FUNCTION "FC_RouteFSM" : Void
{ S7_Optimized_Access := 'TRUE' }
VERSION : 4.6
// ==============================================================================
// FC_RouteFSM - Керування маршрутом (Mailbox Pattern v4.0)
// ==============================================================================
// Версія: 4.6.0
// Дата: 2026-05-15
// ==============================================================================
// ЗМІНИ v4.6.0:
//   [FEAT] Реалізовано "Різкий останов" (Fast Stop) при аварії механізму.
//   [FEAT] Додана детальна перевірка GrainType для ям та силосів.
//   [FIX] Виключено перевірку типу для конкретних силосів (1,2,19,25,26,27).
//   [FEAT] Додано очікування цільової позиції для засувок (Gate2P) та клапанів (Valve3P).
//   [FEAT] Додано очікування цільової позиції для засувок (Gate2P) та клапанів (Valve3P) при пуску та зупинці.
//   [FIX] Виправлено назву константи TYPE_RECEIVING_PIT.
//
// ЗМІНИ v4.0.0:
//   [FIX] RUNNING/STOPPING: затримка (StartDelayMs/StopDelayMs) тепер відбувається
//         ПЕРЕД видачею команди, а не ПІСЛЯ досягнення цільового стану.
//         БУЛО: CMD_START → wait target → IF delay > 0 → pause → advance
//         СТАЛО: IF delay > 0 → pause first → CMD_START → wait target → advance
//         stepPauseTck = 0 означає "новий крок, затримка ще не почалась".
//   [FEAT] Додано підтримку TYPE_FAN та TYPE_FEEDER в CASE для читання затримок.
//   [FIX] Видалено використання RS_TimeoutMs (якого більше немає в UDT_RouteStep).
//         Тепер використовуються індивідуальні затримки з механізмів.
//
// ЗМІНИ v3.9.2:
//   [FIX] STOPPING: advance-блок переписано з явним флагом doAdvance (VAR_TEMP).
//         БУЛО: окремий "NOT stepPause AND stopped" блок — умова могла бути TRUE
//               в циклах де pause ще не виставлена.
//         СТАЛО: doAdvance := TRUE ТІЛЬКИ у двох явних випадках:
//               - Phase A: механізм зупинився AND RS_TimeoutMs = 0
//               - Phase B: таймер спрацював (timeElapsed = TRUE)
//         Симетрично з RUNNING (де advance теж всередині Phase B IF timeElapsed).
//
// ЗМІНИ v3.9.1:
//   [FIX] TIA Portal SCL не дозволяє виклик функції з VAR_OUTPUT в IF-виразі.
//         FC_TimeElapsedMs (має VAR_OUTPUT ElapsedMs, NowTck) → результат
//         тепер зберігається у VAR_TEMP timeElapsed : BOOL перед IF.
//         Додано VAR_TEMP секцію.
//
// ЗМІНИ v3.9.0:
//   [FEAT-3] RUNNING: пауза між кроками через RS_TimeoutMs (аналогічно STOPPING).
//            Фаза A: видати команду → чекаємо цільового стану (RUNNING або IDLE).
//            Фаза B (stepPause=TRUE): чекаємо RS_TimeoutMs мс, потім advance.
//            RS_TimeoutMs = 0 → Фаза B відсутня (поведінка як раніше).
//            Перейменовано: stopPause→stepPause, stopPauseTck→stepPauseTck.
//
// ЗМІНИ v3.8.0:
//   [FEAT-2] STOPPING: пауза між кроками через RS_TimeoutMs.
//            Фаза A: CMD_STOP кожен цикл → чекаємо зупинки механізму.
//            Фаза B (stepPause=TRUE): чекаємо RS_TimeoutMs мс після зупинки.
//            RS_TimeoutMs = 0 → Фаза B відсутня (поведінка як у v3.7).
//            Нові поля UDT_RouteFsm: stepPause : BOOL, stepPauseTck : DINT.
//
// ЗМІНИ v3.7.0:
//   [FEAT-1] STOPPING: послідовна зупинка у зворотньому порядку.
//            БУЛО: CMD_STOP до всіх механізмів одночасно (FOR по всіх кроках),
//                  потім очікування allStopped.
//            СТАЛО: зупинка крок-за-кроком від stepCnt до 1 (1-based).
//                   Кожен цикл — CMD_STOP до поточного кроку (RF_ActiveStep).
//                   Коли поточний зупинився → RF_ActiveStep-- → наступний крок.
//                   Коли крок 1 зупинився → CMD_RELEASE_OWNER для всіх → ABORTED.
//            RF_ActiveStep ініціалізується = stepCnt при вході з RUNNING (1-based).
//
// ЗМІНИ v3.6.2:
//   [FIX-12] VALIDATING: додано перевірку сумісності RS_Action + RS_Wait.
//            RS_ACT_STOP + RS_WAIT_RUNNING → ROUTE_REJ_BY_CONTRACT.
//            До виправлення: ця комбінація проходила валідацію, але у RUNNING
//            механізм після CMD_STOP ніколи не досягав STS_RUNNING →
//            крок зависав нескінченно (до зовнішнього fault або SafetyStop).
//
// ЗМІНИ v3.6.1:
//   [FIX-10] Ранній скан anyFault/anyLocal + GlobalSafetyStop блок:
//            додано IF slot > MECHS_COUNT THEN CONTINUE перед Mechs[slot].
//            До виправлення: у першому циклі нової команди з невалідним RS_Slot
//            обидва цикли зверталися до Mechs[invalid] до того, як VALIDATING
//            встигав відхилити крок → потенційний OOB і зупинка CPU (OB121).
//
// ЗМІНИ v3.6.0:
//   [FIX-8] Виправлено хибний коментар у STOPPING → CMD_RELEASE_OWNER.
//           БУЛО:   "STS_DISABLED → OwnerCur вже NONE → ARB_OWNER_BUSY"
//           ФАКТ:   OwnerCur залишається OWNER_ROUTE після переходу у STS_DISABLED
//                   (механізм не скидає OwnerCur самостійно).
//                   CMD_RELEASE_OWNER → ARB_WRONG_STATUS (DISABLED ≠ IDLE/FAULT).
//                   dummyOk → ABORTED → retry кожен цикл → Enable_OK відновлено
//                   → STS_IDLE → ARB_OK → звільнено ✓   (FIX-5 зберігає StepCount).
//
//   [FIX-9] Видалено недосяжний код у VALIDATING (перевірка startEdge).
//           startEdge завжди FALSE у циклі VALIDATING:
//             Цикл N (IDLE):       lastCmd=RT_CMD_NONE → startEdge=TRUE → lastCmd:=RT_CMD_START
//             Цикл N+1 (VALID.):   lastCmd=RT_CMD_START, Cmd=RT_CMD_START → startEdge=FALSE
//           Supervisor блокує новий START поки isActive → RouteExecutor не змінюється.
//           Константа ROUTE_REJ_DUPLICATE_START більше не використовується.
//
// ЗМІНИ v3.5.0:
//   [FIX-7] ABORTED/REJECTED: startEdge → прямий перехід у VALIDATING.
//
//           ПРОБЛЕМА: маршрут у ABORTED, SCADA надсилає RT_CMD_START.
//           Цикл N:   Supervisor копіює START → RouteExecutor (processedRouteId захищає).
//                     FSM ABORTED: RC_Cmd ≠ RT_CMD_NONE → лишається ABORTED.
//           Цикл N+1: Cleanup бачить ABORTED + allReleased → RC_Cmd=RT_CMD_NONE, StepCount=0.
//                     FSM ABORTED: RT_CMD_NONE → IDLE.
//           Цикл N+2: FSM IDLE: RC_Cmd=RT_CMD_NONE → startEdge=FALSE → нічого.
//           START мовчки загублено.
//
//           РІШЕННЯ: у ABORTED/REJECTED перевіряємо startEdge першим.
//           Якщо startEdge → VALIDATING (скидаємо ResultCode/ActiveStep/StepSts).
//           Цикл N+1: стан вже VALIDATING → Cleanup не чіпає → кроки збережені ✓
//           Механізми ще OWNER_ROUTE (ABORTED-retry) → VALIDATING відкидає REJ_BY_OWNER
//           (коректна поведінка; оператор бачить REJECTED, а не мовчазний IDLE).
//
// ЗМІНИ v3.4.0:
//   - VALIDATING: додано перевірку RS_Slot > MECHS_COUNT → ROUTE_REJ_BY_CONTRACT.
//   - Захист від виходу за межі масиву Mechs[] при невалідному слоті від SCADA.
//   - Перевірка стоїть першою у циклі — до будь-якого звернення до Mechs[slot].
//   - Всі наступні стани (STARTING/RUNNING/STOPPING) отримують гарантовано валідний слот.
//
// ==============================================================================
// ЗМІНИ v3.0.0:
//   - FC_ArbiterMech: повертає USINT (RejectCode) замість BOOL
//   - CMD_NONE заборонено → CMD_SET_OWNER_SCADA / CMD_RELEASE_OWNER
//   - lockOkOne, cmdOk, dummyOk: BOOL → USINT у UDT_RouteFsm
//
// ЗМІНИ v3.1.0:
//   - ABORTED: retry CMD_RELEASE_OWNER кожен цикл поки OwnerCur = OWNER_ROUTE
//   - Вирішує застряглий ownership після GlobalSafetyStop
//
// ЗМІНИ v3.2.0:
//   - STOPPING: виправлено allStopped — рахує STS_FAULT/DISABLED/LOCAL як зупинені
//   - БУЛО:   Status <> STS_IDLE → не зупинений
//   - СТАЛО:  Status IN {STARTING, RUNNING, STOPPING} → не зупинений
//
// ЗМІНИ v3.3.0:
//   - GlobalSafetyStop: ДОДАНО CMD_STOP перед CMD_RELEASE_OWNER
//   - БУЛО: тільки CMD_RELEASE_OWNER (best effort) → мотор міг крутитись ~2 сек
//   - СТАЛО: спочатку CMD_STOP (наказ зупинитись), потім CMD_RELEASE_OWNER
//   - Тепер механізм отримує команду зупинки негайно і йде STS_STOPPING→STS_IDLE
//     замість чекати SpeedLost timeout → STS_FAULT
//   - CMD_RELEASE_OWNER після CMD_STOP все одно може повернути ARB_WRONG_STATUS
//     (механізм ще RUNNING/STOPPING), retry відбувається у ABORTED як раніше
//
// ГАРАНТІЇ ЗУПИНКИ:
//   Нормальний STOP_OP:
//     STOPPING: CMD_STOP кожен цикл → STS_STOPPING→STS_IDLE →
//     allStopped → CMD_RELEASE_OWNER (ARB_OK) → ABORTED ✓
//
//   Аварія під час зупинки (STOPPING):
//     STS_FAULT → allStopped (FAULT рахується) →
//     CMD_RELEASE_OWNER (ARB_OK, FAULT дозволено) → ABORTED ✓
//
//   Enable_OK знімається під час зупинки (STOPPING):
//     STS_DISABLED + OwnerCur=NONE (механізм сам скинув) → allStopped →
//     CMD_RELEASE_OWNER → ARB_OWNER_BUSY (dummyOk) → ABORTED ✓
//
//   GlobalSafetyStop (механізм у STS_RUNNING):
//     CMD_STOP → Mechs[slot].Cmd=CMD_STOP → механізм → STS_STOPPING
//     CMD_RELEASE_OWNER → ARB_WRONG_STATUS (ще не IDLE) → ABORTED
//     Retry у ABORTED: STS_STOPPING→STS_IDLE → ARB_OK → OwnerCur=NONE ✓
//     (якщо апаратна безпека вбила живлення → STS_FAULT → ARB_OK ✓)
//
// АРХІТЕКТУРА:
//   FC_RouteFSM    — логіка переходів, послідовність кроків
//   FC_ArbiterMech — захоплення ownership, запис команди
//   FC_Noria/...   — виконання команди, зміна Status, аварії
//   FC_Route_Supervisor — Mailbox→RouteExecutor, виклик FSM, cleanup
// ==============================================================================
   VAR_INPUT
      RouteIdx : USInt;   // ID маршруту (1..12)
      Cmd : "UDT_RouteCmd";   // Команда та кроки маршруту
   END_VAR

   VAR_OUTPUT
      Sts : "UDT_RouteStatus";
   END_VAR

   VAR_IN_OUT
      Mechs : Array[0.."MECHS_COUNT"] of "UDT_BaseMechanism";
      Fsm : "UDT_RouteFsm";
   END_VAR

   VAR_TEMP
      timeElapsed : Bool;   // проміжний результат FC_TimeElapsedMs
      elapsedMs : DInt;   // допоміжний вихід FC_TimeElapsedMs (ігнорується)
      nowTck : DInt;   // допоміжний вихід FC_TimeElapsedMs (ігнорується)
      doAdvance : Bool;   // TRUE = виконати advance у STOPPING (після Phase A або Phase B)
      stepDelayMs : DInt;   // індивідуальна затримка з механізму (StartDelayMs/StopDelayMs)
      grainTypePit : Int;   // тип зерна ями (для перевірки сумісності)
      grainTypeSilo : Int;   // тип зерна силосу (для перевірки сумісності)
      firstSiloGrainType : Int;   // тип першого силосу в маршруті
      siloCnt : Int;   // кількість силосів у маршрутi
      siloMissingType : Bool;   // TRUE = один із силосів має незаданий тип
      siloGrainMismatch : Bool;   // TRUE = в маршруті два силоси з різними типами зерна
      isSiloExcluded : Bool;   // TRUE = силос виключений з перевірки GrainType
      forceGrainType : Bool;   // TRUE = силос має Force_Code BIT10 — ігнорувати перевірку GrainType
      hasPit : Bool;   // TRUE = у маршруті є яма
      hasSilo : Bool;   // TRUE = у маршруті є силос
   END_VAR


BEGIN

	// =========================================================
	// Edge detection команд маршруту
	// =========================================================
	#Fsm.startEdge := (#Cmd.RC_Cmd = "RT_CMD_START") AND (#Fsm.lastCmd <> "RT_CMD_START");
	#Fsm.stopOpEdge := (#Cmd.RC_Cmd = "RT_CMD_STOP_OP") AND (#Fsm.lastCmd <> "RT_CMD_STOP_OP");
	#Fsm.lastCmd := #Cmd.RC_Cmd;

	// =========================================================
	// Кількість кроків (з обмеженням)
	// =========================================================
	#Fsm.stepCnt := USINT_TO_INT(#Cmd.RC_StepCount);
	IF #Fsm.stepCnt < 1 THEN
	    #Fsm.stepCnt := 1;
	END_IF;
	IF #Fsm.stepCnt > "ROUTE_MAX_STEPS" THEN
	    #Fsm.stepCnt := "ROUTE_MAX_STEPS";
	END_IF;

	// Захист від неініціалізованого стану
	IF #Fsm.RF_State = 0 THEN
	    #Fsm.RF_State := "ROUTE_STS_IDLE";
	END_IF;

	// =========================================================
	// Сканування механізмів: аварії та LocalManual
	// =========================================================
	#Fsm.anyFault := FALSE;
	#Fsm.anyLocal := FALSE;
	#Fsm.safetyHit := FALSE;

	IF #Fsm.stepCnt > 0 THEN
	    FOR #Fsm.i := 1 TO #Fsm.stepCnt DO
	        #Fsm.slot := #Cmd.RC_Steps[#Fsm.i].RS_Slot;
	        IF #Fsm.slot > "MECHS_COUNT" THEN
	            CONTINUE;
	        END_IF;

	        IF #Mechs[#Fsm.slot].FLTCode <> 0 THEN
	            #Fsm.anyFault := TRUE;
	        END_IF;

	        IF "GlobalLocalManual" OR #Mechs[#Fsm.slot].LocalManual THEN
	            #Fsm.anyLocal := TRUE;
	        END_IF;

	        IF #Fsm.anyFault AND #Fsm.anyLocal THEN
	            EXIT;
	        END_IF;
	    END_FOR;
	END_IF;

	// =========================================================
	// АВАРІЙНА ЗУПИНКА (GlobalSafetyStop) — найвищий пріоритет
	// =========================================================
	// Послідовність для кожного механізму:
	//   1. CMD_STOP       — наказ зупинитись негайно (незалежно від послідовності)
	//                       ARB_OK → Mechs[slot].Cmd = CMD_STOP ✓
	//                       ARB_OWNER_BUSY → не наш механізм, не критично
	//                       ARB_LOCAL_MANUAL → оператор сам відповідає
	//   2. CMD_RELEASE_OWNER — спроба звільнити власника (best effort)
	//                       ARB_WRONG_STATUS якщо ще RUNNING/STOPPING → retry у ABORTED
	//
	// Чому не чекаємо STS_IDLE перед CMD_RELEASE_OWNER:
	//   Safety stop = негайно, без очікування. Механізм зупиниться сам
	//   (STS_STOPPING→STS_IDLE або апаратна безпека→STS_FAULT).
	//   Retry у ABORTED звільнить ownership коли механізм зупиниться.
	// =========================================================
	IF "GlobalSafetyStop" THEN
	    #Fsm.safetyHit := TRUE;

	    IF #Fsm.stepCnt > 0 THEN
	        FOR #Fsm.i := 1 TO #Fsm.stepCnt DO
	            #Fsm.slot := #Cmd.RC_Steps[#Fsm.i].RS_Slot;
	            IF #Fsm.slot > "MECHS_COUNT" THEN
	                CONTINUE;
	            END_IF;

	            // КРОК 1: Зупинити механізм
	            #Fsm.dummyOk := "FC_ArbiterMech"(
	                                             OwnerReq := "OWNER_ROUTE",
	                                             OwnerReqId := USINT_TO_UINT(#RouteIdx),
	                                             ReqCmd := "CMD_STOP",
	                                             ReqParam1 := 0,
	                                             M := #Mechs[#Fsm.slot]
	            );

	            // КРОК 2: Звільнити власника (best effort)
	            // Якщо STS_RUNNING/STOPPING → ARB_WRONG_STATUS → retry у ABORTED
	            #Fsm.dummyOk := "FC_ArbiterMech"(
	                                             OwnerReq := "OWNER_ROUTE",
	                                             OwnerReqId := USINT_TO_UINT(#RouteIdx),
	                                             ReqCmd := "CMD_RELEASE_OWNER",
	                                             ReqParam1 := 0,
	                                             M := #Mechs[#Fsm.slot]
	            );

	        END_FOR;
	    END_IF;

	    #Fsm.RF_State := "ROUTE_STS_ABORTED";
	    #Fsm.RF_ResultCode := "ROUTE_ABRT_BY_SAFETY";
	END_IF;

	// =========================================================
	// FSM маршруту
	// =========================================================
	IF NOT #Fsm.safetyHit THEN

	    // --------------------------------------------------------
	    // IDLE
	    // --------------------------------------------------------
	    IF #Fsm.RF_State = "ROUTE_STS_IDLE" THEN

	        IF #Fsm.startEdge THEN
	            #Fsm.RF_ResultCode := 0;
	            #Fsm.RF_AbortLatched := 0;
	            #Fsm.RF_ActiveStep := 1;  // 1-based: перший крок [1]
	            #Fsm.RF_StepSts := "STEP_STS_IDLE";
	            #Fsm.RF_State := "ROUTE_STS_VALIDATING";
	        END_IF;

	        // --------------------------------------------------------
	        // VALIDATING
	        // --------------------------------------------------------
	    ELSIF #Fsm.RF_State = "ROUTE_STS_VALIDATING" THEN

	        IF #Fsm.stepCnt <= 0 THEN
	            #Fsm.RF_State := "ROUTE_STS_REJECTED";
	            #Fsm.RF_ResultCode := "ROUTE_REJ_BY_CONTRACT";

	        ELSE
	            FOR #Fsm.i := 1 TO #Fsm.stepCnt DO
	                #Fsm.slot := #Cmd.RC_Steps[#Fsm.i].RS_Slot;
	                #Fsm.stepOk := TRUE;

	                // Сушилка не керується маршрутом — скіп
	                IF #Fsm.slot <= "MECHS_COUNT" THEN
	                    IF #Mechs[#Fsm.slot].DeviceType = "TYPE_SUSHKA" THEN
	                        CONTINUE;
	                    END_IF;
	                END_IF;

	                // Контракт: RS_Slot (перша перевірка — до будь-якого Mechs[slot])
	                IF #Fsm.slot > "MECHS_COUNT" THEN
	                    #Fsm.stepOk := FALSE;
	                END_IF;

	                // Контракт: RS_Action
	                IF (#Cmd.RC_Steps[#Fsm.i].RS_Action <> "RS_ACT_START")
	                    AND (#Cmd.RC_Steps[#Fsm.i].RS_Action <> "RS_ACT_STOP") THEN
	                    #Fsm.stepOk := FALSE;
	                END_IF;

	                // Контракт: RS_Wait
	                IF (#Cmd.RC_Steps[#Fsm.i].RS_Wait <> "RS_WAIT_RUNNING")
	                    AND (#Cmd.RC_Steps[#Fsm.i].RS_Wait <> "RS_WAIT_STOPPED") THEN
	                    #Fsm.stepOk := FALSE;
	                END_IF;

	                // Контракт: RS_Action + RS_Wait сумісність
	                // RS_ACT_STOP + RS_WAIT_RUNNING: після CMD_STOP механізм іде
	                // STOPPING→IDLE і ніколи не повернеться у STS_RUNNING →
	                // крок ніколи не завершиться → маршрут зависає в RUNNING.
	                IF (#Cmd.RC_Steps[#Fsm.i].RS_Action = "RS_ACT_STOP")
	                    AND (#Cmd.RC_Steps[#Fsm.i].RS_Wait = "RS_WAIT_RUNNING") THEN
	                    #Fsm.stepOk := FALSE;
	                END_IF;

	                IF NOT #Fsm.stepOk THEN
	                    #Fsm.RF_State := "ROUTE_STS_REJECTED";
	                    #Fsm.RF_ResultCode := "ROUTE_REJ_BY_CONTRACT";
	                    EXIT;

	                ELSIF #Mechs[#Fsm.slot].OwnerCur <> "OWNER_NONE" THEN
	                    #Fsm.RF_State := "ROUTE_STS_REJECTED";
	                    #Fsm.RF_ResultCode := "ROUTE_REJ_BY_OWNER";
	                    EXIT;

	                ELSIF (NOT #Mechs[#Fsm.slot].Enable_OK)
	                    OR "GlobalLocalManual"
	                    OR #Mechs[#Fsm.slot].LocalManual
	                    OR (#Mechs[#Fsm.slot].FLTCode <> 0) THEN
	                    #Fsm.RF_State := "ROUTE_STS_REJECTED";
	                    #Fsm.RF_ResultCode := "ROUTE_REJ_NOT_READY";
	                    EXIT;
	                END_IF;

	            END_FOR;

	            IF #Fsm.RF_State = "ROUTE_STS_VALIDATING" THEN
	                // Перевірка GrainType: яма і силос повинні мати однаковий ненульовий тип,
	                // а якщо в маршруті два силоси — їхні типи також повинні співпадати.
	                #grainTypePit := 0;
	                #grainTypeSilo := 0;
	                #firstSiloGrainType := 0;
	                #siloCnt := 0;
	                #siloMissingType := FALSE;
	                #siloGrainMismatch := FALSE;
	                #isSiloExcluded := FALSE;
	                #forceGrainType := FALSE;
	                #hasPit := FALSE;
	                #hasSilo := FALSE;

	                FOR #Fsm.i := 1 TO #Fsm.stepCnt DO
	                    #Fsm.slot := #Cmd.RC_Steps[#Fsm.i].RS_Slot;
	                    IF #Fsm.slot <= "MECHS_COUNT" THEN
	                        IF #Mechs[#Fsm.slot].DeviceType = "TYPE_RECEIVING_PIT" THEN
	                            #hasPit := TRUE;
	                            #grainTypePit := "DB_Mechs".ReceivingPit[#Mechs[#Fsm.slot].TypedIndex].GrainType;
	                        ELSIF #Mechs[#Fsm.slot].DeviceType = "TYPE_SILOS" THEN
	                            #hasSilo := TRUE;
	                            // Исключения: силосы с TypedIndex 1,2,19,25,26,27 не проверяем GrainType
	                            #isSiloExcluded := (#Mechs[#Fsm.slot].TypedIndex = 1 OR #Mechs[#Fsm.slot].TypedIndex = 2 OR
	                            #Mechs[#Fsm.slot].TypedIndex = 19 OR #Mechs[#Fsm.slot].TypedIndex = 25 OR
	                            #Mechs[#Fsm.slot].TypedIndex = 26 OR #Mechs[#Fsm.slot].TypedIndex = 27);
	                            IF NOT #isSiloExcluded THEN
	                                #siloCnt := #siloCnt + 1;
	                                #grainTypeSilo := "DB_Mechs".Silos[#Mechs[#Fsm.slot].TypedIndex].GrainType;
	                                IF #grainTypeSilo = 0 THEN
	                                    #siloMissingType := TRUE;
	                                END_IF;
	                                IF #siloCnt = 1 THEN
	                                    #firstSiloGrainType := #grainTypeSilo;
	                                ELSIF #firstSiloGrainType <> #grainTypeSilo THEN
	                                    #siloGrainMismatch := TRUE;
	                                END_IF;
	                            END_IF;
	                            IF (#Mechs[#Fsm.slot].Force_Code AND 1024) <> 0 THEN
	                                #forceGrainType := TRUE;
	                            END_IF;
	                        END_IF;
	                    END_IF;
	                END_FOR;

	                IF NOT #forceGrainType THEN
	                    // Силос в маршруті і один із силосів не має заданого типу
	                    IF #hasSilo AND #siloMissingType THEN
	                        #Fsm.RF_State := "ROUTE_STS_REJECTED";
	                        #Fsm.RF_ResultCode := "ROUTE_REJ_GRAIN_NOT_SET";
	                        // Яма в маршруті і її тип = 0
	                    ELSIF #hasPit AND #grainTypePit = 0 THEN
	                        #Fsm.RF_State := "ROUTE_STS_REJECTED";
	                        #Fsm.RF_ResultCode := "ROUTE_REJ_GRAIN_NOT_SET";
	                        // Два силоси в маршруті і їхні типи не співпадають
	                    ELSIF #siloGrainMismatch THEN
	                        #Fsm.RF_State := "ROUTE_STS_REJECTED";
	                        #Fsm.RF_ResultCode := "ROUTE_REJ_SILOS_GRAIN_MISMATCH";
	                        // Обидва (яма + силос) в маршруті і типи не співпадають
	                    ELSIF #hasSilo AND #hasPit AND #firstSiloGrainType <> #grainTypePit THEN
	                        #Fsm.RF_State := "ROUTE_STS_REJECTED";
	                        #Fsm.RF_ResultCode := "ROUTE_REJ_GRAIN_MISMATCH";
	                    END_IF;
	                END_IF;
	            END_IF;

	            IF #Fsm.RF_State = "ROUTE_STS_VALIDATING" THEN
	                #Fsm.RF_State := "ROUTE_STS_STARTING";
	            END_IF;
	        END_IF;

	        // --------------------------------------------------------
	        // STARTING — атомарне захоплення всіх механізмів
	        // --------------------------------------------------------
	    ELSIF #Fsm.RF_State = "ROUTE_STS_STARTING" THEN

	        #Fsm.lockOkAll := TRUE;

	        IF #Fsm.stepCnt > 0 THEN
	            FOR #Fsm.i := 1 TO #Fsm.stepCnt DO
	                #Fsm.slot := #Cmd.RC_Steps[#Fsm.i].RS_Slot;

	                // Сушилка не керується маршрутом — не захоплюємо owner
	                IF #Mechs[#Fsm.slot].DeviceType = "TYPE_SUSHKA" THEN
	                    CONTINUE;
	                END_IF;

	                // CMD_SET_OWNER_SCADA = захопити власника без виконання команди
	                #Fsm.lockOkOne := "FC_ArbiterMech"(
	                                                   OwnerReq := "OWNER_ROUTE",
	                                                   OwnerReqId := USINT_TO_UINT(#RouteIdx),
	                                                   ReqCmd := "CMD_SET_OWNER_SCADA",
	                                                   ReqParam1 := 0,
	                                                   M := #Mechs[#Fsm.slot]
	                );

	                IF #Fsm.lockOkOne <> "ARB_OK" THEN
	                    #Fsm.lockOkAll := FALSE;
	                END_IF;
	            END_FOR;
	        ELSE
	            #Fsm.lockOkAll := FALSE;
	        END_IF;

	        IF NOT #Fsm.lockOkAll THEN
	            // Відкат: звільнити вже захоплені механізми.
	            // Механізми ще у IDLE (не запускались) → CMD_RELEASE_OWNER пройде.
	            // Механізм що не захопився → ARB_OWNER_BUSY → dummyOk.
	            IF #Fsm.stepCnt > 0 THEN
	                FOR #Fsm.i := 1 TO #Fsm.stepCnt DO
	                    #Fsm.slot := #Cmd.RC_Steps[#Fsm.i].RS_Slot;

	                    #Fsm.dummyOk := "FC_ArbiterMech"(
	                                                     OwnerReq := "OWNER_ROUTE",
	                                                     OwnerReqId := USINT_TO_UINT(#RouteIdx),
	                                                     ReqCmd := "CMD_RELEASE_OWNER",
	                                                     ReqParam1 := 0,
	                                                     M := #Mechs[#Fsm.slot]
	                    );
	                END_FOR;
	            END_IF;

	            #Fsm.RF_State := "ROUTE_STS_REJECTED";
	            #Fsm.RF_ResultCode := "ROUTE_REJ_BY_OWNER";

	        ELSE
	            #Fsm.RF_State := "ROUTE_STS_RUNNING";
	        END_IF;

	        // --------------------------------------------------------
	        // RUNNING — виконання кроків по черзі (затримка ПЕРЕД командою)
	        // --------------------------------------------------------
	    ELSIF #Fsm.RF_State = "ROUTE_STS_RUNNING" THEN

	        // --- Умови переривання (перевіряються до виконання кроку) ---
	        IF #Fsm.stopOpEdge THEN
	            #Fsm.RF_AbortLatched := "ROUTE_ABRT_BY_OPERATOR";
	            #Fsm.RF_ActiveStep := INT_TO_USINT(#Fsm.stepCnt);  // 1-based: останній крок [stepCnt]
	            #Fsm.stepPause := FALSE;
	            #Fsm.stepPauseTck := 0;
	            #Fsm.RF_State := "ROUTE_STS_STOPPING";

	        ELSIF #Fsm.anyLocal THEN
	            #Fsm.RF_AbortLatched := "ROUTE_ABRT_BY_LOCAL";
	            #Fsm.RF_ActiveStep := INT_TO_USINT(#Fsm.stepCnt);  // 1-based
	            #Fsm.stepPause := FALSE;
	            #Fsm.stepPauseTck := 0;
	            #Fsm.RF_State := "ROUTE_STS_STOPPING";

	        ELSIF #Fsm.anyFault THEN
	            #Fsm.RF_ResultCode := "ROUTE_ABRT_BY_FAULT";

	            // РЕЗКИЙ ОСТАНОВ: негайно зупинити всі механізми маршруту
	            IF #Fsm.stepCnt > 0 THEN
	                FOR #Fsm.i := 1 TO #Fsm.stepCnt DO
	                    #Fsm.slot := #Cmd.RC_Steps[#Fsm.i].RS_Slot;
	                    IF #Fsm.slot > 0 AND #Fsm.slot <= "MECHS_COUNT" THEN
	                        #Fsm.dummyOk := "FC_ArbiterMech"(
	                            OwnerReq := "OWNER_ROUTE",
	                            OwnerReqId := USINT_TO_UINT(#RouteIdx),
	                            ReqCmd := "CMD_STOP",
	                            ReqParam1 := 0,
	                            M := #Mechs[#Fsm.slot]);
	                    END_IF;
	                END_FOR;
	            END_IF;
	            #Fsm.RF_State := "ROUTE_STS_ABORTED";

	        ELSE
	            // --- Поточний крок ---
	            #Fsm.stepIdx := USINT_TO_INT(#Fsm.RF_ActiveStep);

	            IF #Fsm.stepIdx > #Fsm.stepCnt THEN
	                // Всі кроки виконано — залишаємось у RUNNING.
	                // Механізми залишаються під Owner=ROUTE.
	                // SCADA бачить ResultCode=200 → маршрут активний.
	                #Fsm.RF_ResultCode := "ROUTE_OK_RUNNING";  // BIT15 = 32768

	            ELSE
	                #Fsm.slot := #Cmd.RC_Steps[#Fsm.stepIdx].RS_Slot;

	                // === Читати StartDelayMs з механизма ===
	                CASE #Mechs[#Fsm.slot].DeviceType OF
	                    "TYPE_REDLER":
	                        #stepDelayMs := "DB_Mechs".Redler[#Mechs[#Fsm.slot].TypedIndex].StartDelayMs;
	                    "TYPE_NORIA":
	                        #stepDelayMs := "DB_Mechs".Noria[#Mechs[#Fsm.slot].TypedIndex].StartDelayMs;
	                    "TYPE_SEPARATOR":
	                        #stepDelayMs := "DB_Mechs".Separator[#Mechs[#Fsm.slot].TypedIndex].StartDelayMs;
	                    "TYPE_FAN":
	                        #stepDelayMs := "DB_Mechs".Fan[#Mechs[#Fsm.slot].TypedIndex].StartDelayMs;
	                    "TYPE_FEEDER":
	                        #stepDelayMs := "DB_Mechs".Feeder[#Mechs[#Fsm.slot].TypedIndex].StartDelayMs;
	                    ELSE
	                        #stepDelayMs := 0;
	                END_CASE;

	                // === Фаза: Затримка ПЕРЕД командою ===
	                IF #stepDelayMs > 0 AND #Fsm.stepPauseTck = 0 AND NOT #Fsm.stepPause THEN
	                    #timeElapsed := "FC_TimeElapsedMs"(
	                                                       StartTck := 0,
	                                                       TimeoutMs := 0,
	                                                       ElapsedMs => #elapsedMs,
	                                                       NowTck => #Fsm.stepPauseTck);
	                    #Fsm.stepPause := TRUE;
	                END_IF;

	                IF #Fsm.stepPause THEN
	                    // Чекаємо завершення затримки ПЕРЕД командою
	                    #timeElapsed := "FC_TimeElapsedMs"(
	                                                       StartTck := #Fsm.stepPauseTck,
	                                                       TimeoutMs := #stepDelayMs,
	                                                       ElapsedMs => #elapsedMs,
	                                                       NowTck => #nowTck);
	                    IF #timeElapsed THEN
	                        #Fsm.stepPause := FALSE;
	                    END_IF;
	                END_IF;

	                // === Сушилка: скіп кроку ===
	                IF #Mechs[#Fsm.slot].DeviceType = "TYPE_SUSHKA" THEN
	                    #Fsm.stepPauseTck := 0;
	                    #Fsm.RF_ActiveStep := #Fsm.RF_ActiveStep + 1;
	                    #Fsm.RF_StepSts := "STEP_STS_DONE";
	                ELSE
	                // === Фаза: Видача команди + очікування цілі ===
	                IF NOT #Fsm.stepPause THEN
	                    // Видати команду поточного кроку через арбітр (кожен цикл)
	                    IF #Cmd.RC_Steps[#Fsm.stepIdx].RS_Action = "RS_ACT_START" THEN
	                        #Fsm.cmdOk := "FC_ArbiterMech"(
	                                                       OwnerReq := "OWNER_ROUTE",
	                                                       OwnerReqId := USINT_TO_UINT(#RouteIdx),
	                                                       ReqCmd := "CMD_START",
	                                                       ReqParam1 := #Cmd.RC_Steps[#Fsm.stepIdx].RS_StartParam,
	                                                       M := #Mechs[#Fsm.slot]
	                        );
	                    ELSE
	                        #Fsm.cmdOk := "FC_ArbiterMech"(
	                                                       OwnerReq := "OWNER_ROUTE",
	                                                       OwnerReqId := USINT_TO_UINT(#RouteIdx),
	                                                       ReqCmd := "CMD_STOP",
	                                                       ReqParam1 := 0,
	                                                       M := #Mechs[#Fsm.slot]
	                        );
	                    END_IF;

	                    IF #Fsm.cmdOk <> "ARB_OK" THEN
	                        // Арбітр відхилив команду → аварійна зупинка маршруту
	                        #Fsm.RF_AbortLatched := "ROUTE_ABRT_BY_OWNER";
	                        #Fsm.RF_ActiveStep := INT_TO_USINT(#Fsm.stepCnt);  // 1-based
	                        #Fsm.stepPause := FALSE;
	                        #Fsm.stepPauseTck := 0;
	                        #Fsm.RF_State := "ROUTE_STS_STOPPING";

	                    ELSE
	                        #Fsm.RF_StepSts := "STEP_STS_WORK";

	                        // Перевірити умову завершення кроку
	                        IF #Cmd.RC_Steps[#Fsm.stepIdx].RS_Wait = "RS_WAIT_RUNNING" THEN
	                            // Стандартна обробка — перевірка STS_RUNNING
	                            IF #Mechs[#Fsm.slot].Status = "STS_RUNNING" THEN
	                                #Fsm.stepPauseTck := 0;
	                                #Fsm.RF_ActiveStep := #Fsm.RF_ActiveStep + 1;
	                                #Fsm.RF_StepSts := "STEP_STS_DONE";
	                            END_IF;
	                        ELSE  // RS_WAIT_STOPPED
                            // Для засувок та клапанів перевіряємо досягнення цільової позиції
                            IF (#Mechs[#Fsm.slot].DeviceType = "TYPE_GATE2P" OR #Mechs[#Fsm.slot].DeviceType = "TYPE_VALVE3P") THEN
                                IF (#Mechs[#Fsm.slot].Status = "STS_IDLE") AND (#Mechs[#Fsm.slot].Status_Param = #Cmd.RC_Steps[#Fsm.stepIdx].RS_StartParam) THEN
                                    #Fsm.stepPauseTck := 0;
                                    #Fsm.RF_ActiveStep := #Fsm.RF_ActiveStep + 1;
                                    #Fsm.RF_StepSts := "STEP_STS_DONE";
                                END_IF;
                            ELSE
                                IF #Mechs[#Fsm.slot].Status = "STS_IDLE" THEN
                                    #Fsm.stepPauseTck := 0;
                                    #Fsm.RF_ActiveStep := #Fsm.RF_ActiveStep + 1;
                                    #Fsm.RF_StepSts := "STEP_STS_DONE";
                                END_IF;
                            END_IF;
	                        END_IF;
	                    END_IF;
	                END_IF;
	                END_IF; // TYPE_SUSHKA skip (RUNNING)
	            END_IF;
	        END_IF;

	        // --------------------------------------------------------
	        // STOPPING — покрокова зупинка у зворотньому порядку (затримка ПЕРЕД командою)
	        // --------------------------------------------------------
	        // RF_ActiveStep = поточний крок зупинки (stepCnt → 1).
	        // Ініціалізується при вході з RUNNING (= stepCnt).
	        //
	        // Для кожного кроку:
	        //   1. Затримка ПЕРЕД командою (StopDelayMs з механизма):
	        //      stepPauseTck = 0 → почати затримку
	        //      stepPause = TRUE → чекати завершення
	        //      Затримка завершена → stepPause = FALSE
	        //   2. Видача команди STOP + очікування зупинки:
	        //      CMD_STOP кожен цикл → чекаємо поки Status NOT IN {STARTING, RUNNING, STOPPING}
	        //      Зупинився → doAdvance := TRUE
	        //
	        //   Advance (doAdvance=TRUE):
	        //     stepIdx > 1 → RF_ActiveStep-- (наступний крок)
	        //     stepIdx = 1 → CMD_RELEASE_OWNER для всіх → ABORTED
	        //
	        // "Зупинений": STS_IDLE / STS_FAULT / STS_DISABLED / STS_LOCAL
	        // "НЕ зупинений": STS_STARTING / STS_RUNNING / STS_STOPPING
	        // --------------------------------------------------------
	    ELSIF #Fsm.RF_State = "ROUTE_STS_STOPPING" THEN
	        // Якщо під час планової зупинки сталася аварія — переходимо на різкий останов
	        IF #Fsm.anyFault THEN
	            #Fsm.RF_ResultCode := "ROUTE_ABRT_BY_FAULT";
	            FOR #Fsm.i := 1 TO #Fsm.stepCnt DO
	                #Fsm.slot := #Cmd.RC_Steps[#Fsm.i].RS_Slot;
	                IF #Fsm.slot > 0 AND #Fsm.slot <= "MECHS_COUNT" THEN
	                    #Fsm.dummyOk := "FC_ArbiterMech"(
	                        OwnerReq := "OWNER_ROUTE",
	                        OwnerReqId := USINT_TO_UINT(#RouteIdx),
	                        ReqCmd := "CMD_STOP",
	                        ReqParam1 := 0,
	                        M := #Mechs[#Fsm.slot]);
	                END_IF;
	            END_FOR;
	            #Fsm.RF_State := "ROUTE_STS_ABORTED";

	        ELSIF #Fsm.stepCnt > 0 THEN
	            #Fsm.stepIdx := USINT_TO_INT(#Fsm.RF_ActiveStep);
	            #Fsm.slot := #Cmd.RC_Steps[#Fsm.stepIdx].RS_Slot;

	            // === Читати StopDelayMs з механизма ===
	            CASE #Mechs[#Fsm.slot].DeviceType OF
	                "TYPE_REDLER":
	                    #stepDelayMs := "DB_Mechs".Redler[#Mechs[#Fsm.slot].TypedIndex].StopDelayMs;
	                "TYPE_NORIA":
	                    #stepDelayMs := "DB_Mechs".Noria[#Mechs[#Fsm.slot].TypedIndex].StopDelayMs;
	                "TYPE_SEPARATOR":
	                    #stepDelayMs := "DB_Mechs".Separator[#Mechs[#Fsm.slot].TypedIndex].StopDelayMs;
	                "TYPE_FAN":
	                    #stepDelayMs := "DB_Mechs".Fan[#Mechs[#Fsm.slot].TypedIndex].StopDelayMs;
	                "TYPE_FEEDER":
	                    #stepDelayMs := "DB_Mechs".Feeder[#Mechs[#Fsm.slot].TypedIndex].StopDelayMs;
	                ELSE
	                    #stepDelayMs := 0;
	            END_CASE;

	            #doAdvance := FALSE;

	            // === Сушилка: скіп кроку при зупинці ===
	            IF #Mechs[#Fsm.slot].DeviceType = "TYPE_SUSHKA" THEN
	                #doAdvance := TRUE;
	            ELSE
	            // === Фаза: Затримка ПЕРЕД командою ===
	            IF #stepDelayMs > 0 AND #Fsm.stepPauseTck = 0 AND NOT #Fsm.stepPause THEN
	                #timeElapsed := "FC_TimeElapsedMs"(
	                                                   StartTck := 0,
	                                                   TimeoutMs := 0,
	                                                   ElapsedMs => #elapsedMs,
	                                                   NowTck => #Fsm.stepPauseTck);
	                #Fsm.stepPause := TRUE;
	            END_IF;

	            IF #Fsm.stepPause THEN
	                // Чекаємо завершення затримки ПЕРЕД командою
	                #timeElapsed := "FC_TimeElapsedMs"(
	                                                   StartTck := #Fsm.stepPauseTck,
	                                                   TimeoutMs := #stepDelayMs,
	                                                   ElapsedMs => #elapsedMs,
	                                                   NowTck => #nowTck);
	                IF #timeElapsed THEN
	                    #Fsm.stepPause := FALSE;
	                END_IF;
	            END_IF;

	            // === Фаза: Видача команди STOP + очікування зупинки ===
	            IF NOT #Fsm.stepPause THEN
	                // Видача команди зупинки (кожен цикл)
	                IF #Cmd.RC_Steps[#Fsm.stepIdx].RS_StopParam <> 0 THEN
	                    // Параметрична зупинка (напр., засувка у позицію CLOSED)
	                    #Fsm.dummyOk := "FC_ArbiterMech"(
	                                                     OwnerReq := "OWNER_ROUTE",
	                                                     OwnerReqId := USINT_TO_UINT(#RouteIdx),
	                                                     ReqCmd := "CMD_START",
	                                                     ReqParam1 := #Cmd.RC_Steps[#Fsm.stepIdx].RS_StopParam,
	                                                     M := #Mechs[#Fsm.slot]
	                    );
	                ELSE
	                    #Fsm.dummyOk := "FC_ArbiterMech"(
	                                                     OwnerReq := "OWNER_ROUTE",
	                                                     OwnerReqId := USINT_TO_UINT(#RouteIdx),
	                                                     ReqCmd := "CMD_STOP",
	                                                     ReqParam1 := 0,
	                                                     M := #Mechs[#Fsm.slot]
	                    );
	                END_IF;

	                // Перевірка: чи поточний механізм зупинився
	                IF (#Mechs[#Fsm.slot].Status <> "STS_STARTING")
	                    AND (#Mechs[#Fsm.slot].Status <> "STS_RUNNING")
	                    AND (#Mechs[#Fsm.slot].Status <> "STS_STOPPING") THEN

                    // Для засувок та клапанів перевіряємо досягнення цільової позиції при зупинці
                    IF (#Mechs[#Fsm.slot].DeviceType = "TYPE_GATE2P" OR #Mechs[#Fsm.slot].DeviceType = "TYPE_VALVE3P")
                        AND (#Cmd.RC_Steps[#Fsm.stepIdx].RS_StopParam <> 0) THEN

                        IF #Mechs[#Fsm.slot].Status_Param = #Cmd.RC_Steps[#Fsm.stepIdx].RS_StopParam THEN
                            #doAdvance := TRUE;
                        END_IF;
                    ELSE
                        #doAdvance := TRUE;
                    END_IF;
	                END_IF;
	            END_IF;
	            END_IF; // TYPE_SUSHKA skip (STOPPING)

	            // ── Advance ───────────────────────────────────────────────────
	            IF #doAdvance THEN
	                IF #Fsm.stepIdx > 1 THEN
	                    // Перейти до попереднього кроку
	                    #Fsm.RF_ActiveStep := #Fsm.RF_ActiveStep - 1;
	                    #Fsm.stepPauseTck := 0;  // reset для наступного кроку

	                ELSE
	                    // Всі механізми зупинено → CMD_RELEASE_OWNER + ABORTED
	                    FOR #Fsm.i := 1 TO #Fsm.stepCnt DO
	                        #Fsm.slot := #Cmd.RC_Steps[#Fsm.i].RS_Slot;
	                        #Fsm.dummyOk := "FC_ArbiterMech"(
	                                                         OwnerReq := "OWNER_ROUTE",
	                                                         OwnerReqId := USINT_TO_UINT(#RouteIdx),
	                                                         ReqCmd := "CMD_RELEASE_OWNER",
	                                                         ReqParam1 := 0,
	                                                         M := #Mechs[#Fsm.slot]
	                        );
	                    END_FOR;

	                    IF #Fsm.RF_AbortLatched = 0 THEN
	                        #Fsm.RF_AbortLatched := "ROUTE_ABRT_BY_OPERATOR";
	                    END_IF;
	                    #Fsm.RF_ResultCode := #Fsm.RF_AbortLatched;
	                    #Fsm.RF_State := "ROUTE_STS_ABORTED";
	                END_IF;
	            END_IF;

	        ELSE
	            // stepCnt = 0 (не повинно траплятись після STARTING) → відразу ABORTED
	            IF #Fsm.RF_AbortLatched = 0 THEN
	                #Fsm.RF_AbortLatched := "ROUTE_ABRT_BY_OPERATOR";
	            END_IF;
	            #Fsm.RF_ResultCode := #Fsm.RF_AbortLatched;
	            #Fsm.RF_State := "ROUTE_STS_ABORTED";
	        END_IF;

	        // --------------------------------------------------------
	        // REJECTED / ABORTED
	        // --------------------------------------------------------
	    ELSIF (#Fsm.RF_State = "ROUTE_STS_REJECTED")
	        OR (#Fsm.RF_State = "ROUTE_STS_ABORTED") THEN

	        // ---------------------------------------------------------
	        // RETRY CMD_RELEASE_OWNER — вирішення застряглого ownership.
	        //
	        // Типовий сценарій після GlobalSafetyStop:
	        //   Цикл N:     CMD_STOP → OK, CMD_RELEASE_OWNER → ARB_WRONG_STATUS
	        //   Цикли N+1..: retry кожен цикл поки механізм зупиняється
	        //   STS_STOPPING → STS_IDLE → ARB_OK → OwnerCur=NONE ✓
	        //   (або апаратна безпека → STS_FAULT → ARB_OK ✓)
	        //
	        // Умова IF: тільки наші механізми (OwnerCur/OwnerCurId перевіряємо).
	        // Якщо вже NONE — умова FALSE, виклик не відбувається.
	        // ---------------------------------------------------------
	        IF #Fsm.stepCnt > 0 THEN
	            FOR #Fsm.i := 1 TO #Fsm.stepCnt DO
	                #Fsm.slot := #Cmd.RC_Steps[#Fsm.i].RS_Slot;

	                IF (#Mechs[#Fsm.slot].OwnerCur = "OWNER_ROUTE")
	                    AND (#Mechs[#Fsm.slot].OwnerCurId = USINT_TO_UINT(#RouteIdx)) THEN

	                    #Fsm.dummyOk := "FC_ArbiterMech"(
	                                                     OwnerReq := "OWNER_ROUTE",
	                                                     OwnerReqId := USINT_TO_UINT(#RouteIdx),
	                                                     ReqCmd := "CMD_RELEASE_OWNER",
	                                                     ReqParam1 := 0,
	                                                     M := #Mechs[#Fsm.slot]
	                    );
	                    // ARB_OK           → OwnerCur = NONE ✓
	                    // ARB_WRONG_STATUS → ще не IDLE/FAULT, retry наступний цикл
	                END_IF;

	            END_FOR;
	        END_IF;

	        // [FIX-7] Re-start: startEdge → прямо у VALIDATING (без проміжного IDLE).
	        // Supervisor вже скопіював кроки у RouteExecutor (Cleanup захищений processedRouteId).
	        // Якщо механізми ще OWNER_ROUTE (ABORTED-retry не завершено) →
	        //   VALIDATING поверне ROUTE_REJ_BY_OWNER (коректна поведінка).
	        IF #Fsm.startEdge THEN
	            #Fsm.RF_ResultCode := 0;
	            #Fsm.RF_AbortLatched := 0;
	            #Fsm.RF_ActiveStep := 1;  // 1-based: перший крок [1]
	            #Fsm.RF_StepSts := "STEP_STS_IDLE";
	            #Fsm.RF_State := "ROUTE_STS_VALIDATING";

	            // Перехід у IDLE коли Supervisor очистить команду (RT_CMD_NONE)
	        ELSIF #Cmd.RC_Cmd = "RT_CMD_NONE" THEN
	            #Fsm.RF_State := "ROUTE_STS_IDLE";
	        END_IF;

	    ELSE
	        // Невідомий стан — скидаємо
	        #Fsm.RF_State := "ROUTE_STS_IDLE";
	    END_IF;

	END_IF;

	// =========================================================
	// Вихідний статус
	// =========================================================
	#Sts.RS_State := #Fsm.RF_State;
	#Sts.RS_ResultCode := #Fsm.RF_ResultCode;
	#Sts.RS_ActiveStep := #Fsm.RF_ActiveStep;
	#Sts.RS_StepSts := #Fsm.RF_StepSts;

END_FUNCTION
